// Mitsubishi GX Works2 project: 模拟工厂工件计数   PLC: FX3U/FX3UC

PROGRAM MAIN
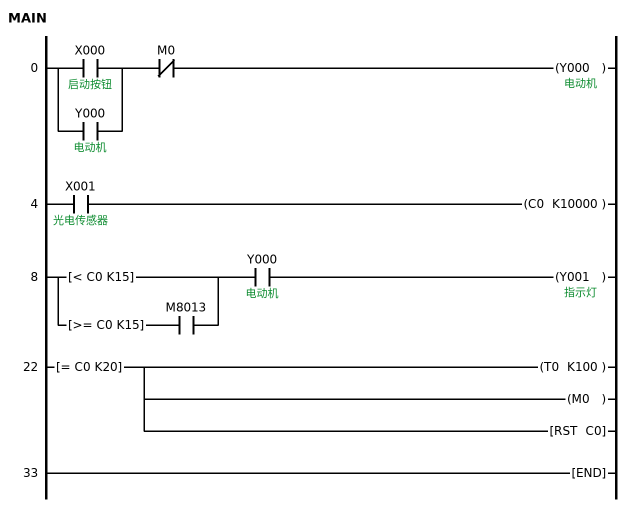
0     LD      X000  ; 启动按钮
      OR      Y000  ; 电动机
      ANI     M0
      OUT     Y000  ; 电动机
4     LD      X001  ; 光电传感器
      OUT     C0 K10000
8     LD<     C0 K15
      LD>=    C0 K15
      AND     M8013
      ORB
      AND     Y000  ; 电动机
      OUT     Y001  ; 指示灯
22    LD=     C0 K20
      OUT     T0 K100
      OUT     M0
      RST     C0
33    END
END_PROGRAM
